FUNCTION_BLOCK MultiAnalog (* Composite Function Block Type *)
  (* Standard: 61499-2 *)
  (* Version 0.0, 3/4/2026, Schneider Electric, template *)
  PACKAGE SE.Nereda;
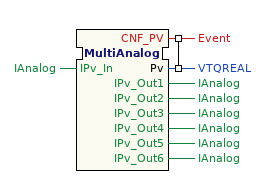
  EVENT_OUTPUT
    CNF_PV WITH Pv; (* Request for new value and limits *)
  END_EVENT
  VAR_OUTPUT
    Pv : VTQREAL; (* Vtq value *)
  END_VAR
  SOCKETS
    IPv_In : IAnalog;
  END_SOCKETS
  PLUGS
    IPv_Out1 : IAnalog;
    IPv_Out2 : IAnalog;
    IPv_Out3 : IAnalog;
    IPv_Out4 : IAnalog;
    IPv_Out5 : IAnalog;
    IPv_Out6 : IAnalog;
  END_PLUGS
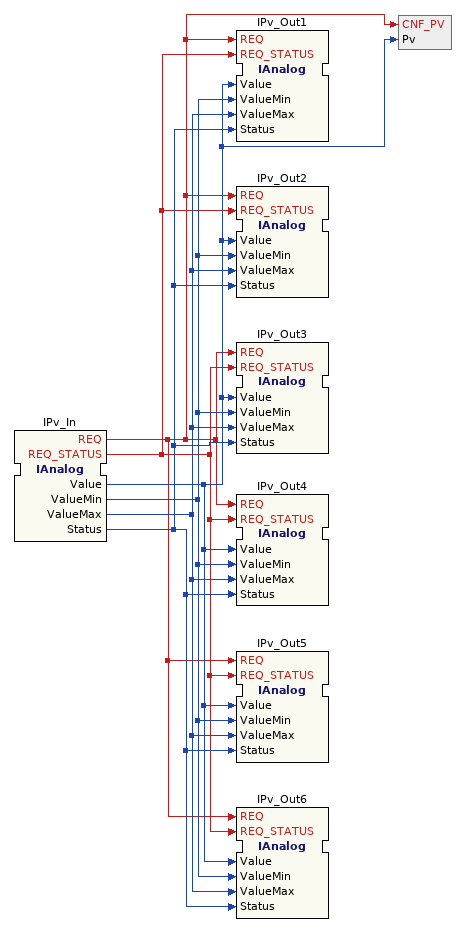
  EVENT_CONNECTIONS
    IPv_In.REQ TO IPv_Out1.REQ;
    IPv_In.REQ TO IPv_Out2.REQ;
    IPv_In.REQ TO IPv_Out3.REQ;
    IPv_In.REQ TO IPv_Out4.REQ;
    IPv_In.REQ TO IPv_Out5.REQ;
    IPv_In.REQ TO IPv_Out6.REQ;
    IPv_In.REQ_STATUS TO IPv_Out1.REQ_STATUS;
    IPv_In.REQ_STATUS TO IPv_Out2.REQ_STATUS;
    IPv_In.REQ_STATUS TO IPv_Out3.REQ_STATUS;
    IPv_In.REQ_STATUS TO IPv_Out4.REQ_STATUS;
    IPv_In.REQ_STATUS TO IPv_Out5.REQ_STATUS;
    IPv_In.REQ_STATUS TO IPv_Out6.REQ_STATUS;
    IPv_In.REQ TO CNF_PV;
  END_CONNECTIONS
  DATA_CONNECTIONS
    IPv_In.Value TO IPv_Out1.Value;
    IPv_In.Value TO IPv_Out2.Value;
    IPv_In.Value TO IPv_Out3.Value;
    IPv_In.ValueMin TO IPv_Out1.ValueMin;
    IPv_In.ValueMin TO IPv_Out2.ValueMin;
    IPv_In.ValueMin TO IPv_Out3.ValueMin;
    IPv_In.ValueMax TO IPv_Out1.ValueMax;
    IPv_In.ValueMax TO IPv_Out2.ValueMax;
    IPv_In.ValueMax TO IPv_Out3.ValueMax;
    IPv_In.Status TO IPv_Out1.Status;
    IPv_In.Status TO IPv_Out2.Status;
    IPv_In.Status TO IPv_Out3.Status;
    IPv_In.Value TO IPv_Out4.Value;
    IPv_In.Value TO IPv_Out5.Value;
    IPv_In.Value TO IPv_Out6.Value;
    IPv_In.ValueMin TO IPv_Out4.ValueMin;
    IPv_In.ValueMin TO IPv_Out5.ValueMin;
    IPv_In.ValueMin TO IPv_Out6.ValueMin;
    IPv_In.ValueMax TO IPv_Out4.ValueMax;
    IPv_In.ValueMax TO IPv_Out5.ValueMax;
    IPv_In.ValueMax TO IPv_Out6.ValueMax;
    IPv_In.Status TO IPv_Out4.Status;
    IPv_In.Status TO IPv_Out5.Status;
    IPv_In.Status TO IPv_Out6.Status;
    IPv_In.Value TO Pv;
  END_CONNECTIONS
END_FUNCTION_BLOCK
